TYPE ST_BaseEvents_Definition :
STRUCT
	uiIDEvent								: UINT;						//unikalny numer zgloszenia dla całego projektu nadawany automatycznie 
	uiIDInItem								: UINT;						//unikalny numer w elemencie - ustawiany podczas dodawania zgłoszenia DO elementu
	bIgnoreRepetitions						: BOOL;						//jak true nie zliczaj powtorzeń wystapienia np komunikaty - alarmy 
	uiRepetitionCounter						: UINT;						//licznik powtórzeń po którym ma się zgłosic błąd
	eEventCategory							: E_BaseEvents_Category;	//BYTE;	//1 - blad, 2 - ostrzezenie, 3 - wiadomosc, 4 - safety
	stDescription							: ST_BaseLabel;
	bConfirm								: BOOL;						// w przypadków niektórych zgłoszeń żeby błąd został skasowany należy go zatwierdzić że operator go zobaczył
END_STRUCT
END_TYPE

(* stored: Version 1.1.0.1
   DUT ST_BaseEvents_Definition: Id {206090b8-93e6-4789-be56-c849744b8cd4} *)
